TYPE T_Ctrl_SIf_IBH_Par :
STRUCT
END_STRUCT
END_TYPE

(* stored: Version 1.1.0.1, ProductVersion 3.1.0.25
   DUT T_Ctrl_SIf_IBH_Par: Id {2385c5e1-2d66-4293-889c-a2e2f1275f64} *)
